SUBAPPLICATION Ventilsteuerung_Uebung_004b2 (* Toggle Flip-Flop mit IE / Split / doppelt *)
  (* Standard: 61499-2 *)
  (* Version 1.0, 2023-10-23, franz *)
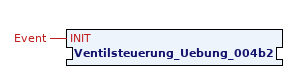
  EVENT_INPUT
    INIT;
  END_EVENT
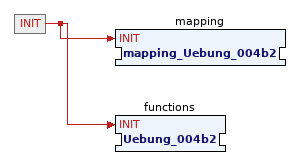
  SUBAPPS
    mapping : mapping_Uebung_004b2;
    functions : Uebung_004b2;
  END_SUBAPPS
  EVENT_CONNECTIONS
    INIT TO mapping.INIT;
    INIT TO functions.INIT;
  END_CONNECTIONS
END_SUBAPPLICATION
